Universal Robots PolyScope program: c_full_bow.urp

Program c_full_bow (installation=string_planes directory=/programs createdIn=5.17.3 lastSavedIn=5.17.3 robotSerialNumber=20245501435)
Calibrated DH parameters: a=[0.000154, -0.137004, -0.385524, -0.00002, 0.000092, 0]; d=[0.162441, 211.794786, -230.585024, 18.923638, 0.099786, 0.09951]; alpha=[1.569493, -0.001902, 0.003874, 1.570111, -1.570167, 0]; deltaTheta=[0, -1.242934, 1.056292, 0.186646, 0.000002, 0.000001]
InitVariablesNode
Robot Program (runOnlyOnce=false)
  bow_dir := True
  note_dur := 1
  Timer (action=Start) variable(name=timer_1)
  If bow_dir≟ True
    MoveL speed 250 mm/s, acceleration 1200 mm/s^2 (useActiveTCP=true) feature=Base
      Waypoint Waypoint_6: TCP in base x=152.636 y=275.824 z=-5.984 mm, rx=-1.6122 ry=-1.6008 rz=0.7404 rad; joints [-153.501, -26.653, 138.52, -151.348, -62.645, -165.795] deg; TCP offset x=28.21 y=-96.107 z=-99.69 mm, rx=0 ry=0 rz=0 rad
        Until EXPRESSION (allowActions=false) ExpressionBranch=timer_1≟note_dur
  Else 
    MoveL speed 250 mm/s, acceleration 1200 mm/s^2 (useActiveTCP=true) feature=Base
      Waypoint Waypoint_4: TCP in base x=245.284 y=570.71 z=53.266 mm, rx=-1.8425 ry=-1.3918 rz=0.0687 rad; joints [-132.226, -24.798, 96.314, -169.322, -42.692, -112.607] deg
        Until EXPRESSION (allowActions=false) ExpressionBranch=timer_1≟note_dur
  SuppressedNode
    MoveL speed 250 mm/s, acceleration 1200 mm/s^2 (useActiveTCP=true) feature=Base
      Waypoint Waypoint_4: TCP in base x=245.284 y=570.71 z=53.266 mm, rx=-1.8425 ry=-1.3918 rz=0.0687 rad; joints [-132.226, -24.798, 96.314, -169.322, -42.692, -112.607] deg
      Waypoint Waypoint_1: TCP in base x=195.249 y=411.456 z=21.268 mm, rx=-1.7342 ry=-1.5169 rz=0.4322 rad; joints [-140.231, -30.936, 122.536, -154.99, -45.802, -143.197] deg
      Waypoint Waypoint_6: TCP in base x=152.636 y=275.824 z=-5.984 mm, rx=-1.6122 ry=-1.6008 rz=0.7404 rad; joints [-153.501, -26.653, 138.52, -151.348, -62.645, -165.795] deg
  Timer (action=Stop) variable=timer_1
  Timer (action=Reset) variable=timer_1
